FUNCTION_BLOCK SawmillPosGen
  (* Standard: 61499-2 *)
  (* Version 0.1, 2017-00-27, Hammond, HAMMONDSDESKTOP *)
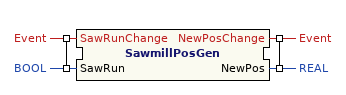
  EVENT_INPUT
    SawRunChange WITH SawRun;
  END_EVENT
  EVENT_OUTPUT
    NewPosChange WITH NewPos;
  END_EVENT
  VAR_INPUT
    SawRun : BOOL;
  END_VAR
  VAR_OUTPUT
    NewPos : REAL;
  END_VAR
  VAR
    PosArrayLen : INT := 20;
    PosArrayPos : INT := 0;
    PosArray : ARRAY [0..19] OF REAL := 0,0.5,1,1.5,2,2.5,3,3.5,4,4.5,5,4.5,4,3.5,3,2.5,2,1.5,1,0.5;
    BusyWork : volatile UDINT := 0;
  END_VAR
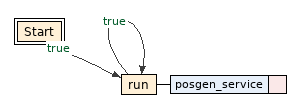
  EC_STATES
    Start;
    run : posgen_service;
  END_STATES
  EC_TRANSITIONS
    Start TO run := true;
    run TO run := true;
  END_TRANSITIONS
  ALGORITHM posgen_service IN C:
//#pragma loopbound min 0 max 2000
//for(me->BusyWork = 0; me->BusyWork < 2000; me->BusyWork++);
if(me->SawRun) {
	me->outputEvents.event.NewPosChange = 1;
	me->NewPos = me->PosArray[me->PosArrayPos];
	me->PosArrayPos++;
	me->PosArrayPos = me->PosArrayPos % me->PosArrayLen;
} else {
	me->outputEvents.event.NewPosChange = 0;
}
  END_ALGORITHM
END_FUNCTION_BLOCK
